TYPE T_Ctrl_SIf_MOD_DtChnToLine :
STRUCT
	dinTest : DINT;
	intDataState : INT;
END_STRUCT
END_TYPE

(* stored: Version 1.1.0.1, ProductVersion 3.1.0.25
   DUT T_Ctrl_SIf_MOD_DtChnToLine: Id {550027d2-1713-423e-8c22-ac70dd31f5c3} *)
